(*			
	EVERDE sp. z o.o.
	Rafał Osajda		22.01.2025		TC 4026.13		wer. 0.0.0.1
	B_Baza dla czujników binarnych styk normalnie otwarty 	
*)
FUNCTION_BLOCK FB_IOSensor_NO EXTENDS FB_IOSensor
VAR
END_VAR

METHOD FB_init : BOOL
VAR_INPUT
	bInitRetains : BOOL; // if TRUE, the retain variables are initialized (warm start / cold start)
	bInCopyCode : BOOL;  // if TRUE, the instance afterwards gets moved into the copy code (online change)
END_VAR
THIS^.eType		:= E_IOSensorType.NO;
END_METHOD

(*			
	EVERDE sp. z o.o.
	Rafał Osajda		05.02.2025		TC 4026.13		wer. 0.0.0.1
	Zwraca aktualny stan czujnika
*)
METHOD IsActive : BOOL
IsActive			:= THIS^.bContact;
END_METHOD

END_FUNCTION_BLOCK

(* stored: Version 1.1.0.1
   POU FB_IOSensor_NO: Id {d281df51-e315-49a9-980a-1299b2b38a3b}, SpecialFunc None
   Method FB_init: Id {0496fef0-cca2-4946-8251-855aeebfd5b6}
   Method IsActive: Id {bf735fd6-b08e-4c2e-aa89-552ead062440} *)
